FUNCTION_BLOCK TestProcess IMPLEMENTS IProcess
VAR
	_running:BOOL := FALSE;
END_VAR

PROPERTY Running : BOOL
GET
Running := _running;
END_GET
END_PROPERTY

METHOD Start
_running := TRUE;
END_METHOD

METHOD Stop
_running := FALSE;
END_METHOD

END_FUNCTION_BLOCK

(* stored: Version 1.1.0.1, ProductVersion 3.1.4024.2
   POU TestProcess: Id {dc01b09e-1521-4822-8420-01f78ff42b6f}, SpecialFunc None
   Property Running: Id {1dbfa749-e7f6-4615-8f07-2406e736e946}
   Get Get: Id {6cf8755d-22a1-4ed2-a3eb-cd4939af4599}
   Method Start: Id {8f82a9ab-c375-44ee-8d67-4910ab883cf1}
   Method Stop: Id {8c8da421-2574-457f-8ab1-66ec70f4c11c} *)
